(* PLC project Tc2_Utilities.TC_Config Demo, tc3-libraries-kb TwinCAT 3.1 *)
(* stored: creationDateTime 2026-05-11T13:00:00, modificationDateTime 2026-05-11T13:00:00 *)

PROGRAM P_Demo_TC_Config
  VAR
    fbTC_Config : TC_Config;  (* TC_Config 实例 *)
    NETID : T_AmsNetId := '';
    SET : BOOL := FALSE;
    TMOUT : TIME := DEFAULT_ADS_TIMEOUT;
    BUSY : BOOL;
    ERR : BOOL;
    ERRID : UDINT;
  END_VAR

// =============================================================================
// 场景：TC_Config 的最小可编译演示——所有 VAR_INPUT 均以 doc/PDF 中真实引脚名调用。
//       业务侧请在线 monitor / 在线写值触发对应输入，看输出端 monitor 结果。
//
// 价值：保证示例 ST 代码所有引脚名与 TC_Config 的 VAR_INPUT/VAR_OUTPUT 一致，
//       Import PLCopenXML → 编译 → 登录 流程能跑通，作为 hand-curated 例程
//       的脚手架。
//
// 验证步骤：
//   1. 引用 Tc2_Utilities（及其依赖 Tc2_System）
//   2. 右键 PLC 项目 → Import PLCopenXML → 选本文件 → OK → 编译、登录
//   3. 在线对 VAR_INPUT 写入合适触发值（典型 bExecute / RUN / START 上升沿）
//   4. 在线 monitor VAR_OUTPUT 观察 FB 反应
// =============================================================================

fbTC_Config(
    NETID := NETID,
    SET := SET,
    TMOUT := TMOUT,
    BUSY => BUSY,
    ERR => ERR,
    ERRID => ERRID
);
END_PROGRAM
